Universal Robots PolyScope program: WORKS.urp

Program WORKS (installation=default directory=/ursim/programs createdIn=5.24.0 lastSavedIn=5.24.0 robotSerialNumber=20195599999)
Calibrated DH parameters: a=[0, -0.425, -0.3922, 0, 0, 0]; d=[0.1625, 0, 0, 0.1333, 0.0997, 0.0996]; alpha=[1.570796, 0, 0, 1.570796, -1.570796, 0]; deltaTheta=[0, 0, 0, 0, 0, 0]
InitVariablesNode
Robot Program (runOnlyOnce=false)
  Wait Sleep waitTime=1
  URCap External Control (External Control, FZI Research Center for Information Technology)
